(* IEC 61131-3 sources: Industry-PLC-LLM/data/PLCBEAD_repo/PLCBEAD_PLCEmbed-main/PLC-BEAD/Source/GEB/building_TIMER_2, 1 file *)

(* ---- TIMER_2.ST ---- *)
FUNCTION UDINT_TO_TIME2:TIME

	VAR_INPUT
		IN :	UDINT;
	END_VAR

	UDINT_TO_TIME2 := DINT_TO_TIME(UDINT_TO_DINT(IN));

END_FUNCTION

FUNCTION_BLOCK T_PLC_MS_block
	VAR_OUTPUT
		T_PLC_MS :	UDINT;
	END_VAR

	VAR
		PLC_TICKS_PER_SEC :	INT;
		PLC_SYS_TICK_CNT :	DINT;
	END_VAR

	VAR
		debug :	BOOL;(*Debug-Mode ON / OFF*)
		N :	INT;(*Debug-Faktor*)
		Offset :	UDINT;(*Debug-Offset*)
		temp :	DWORD := DWORD#1;(*Debug-Offset*)
		MODE :	BOOL;(*modus*)
		faktor :	UDINT;(*Systemtakt-Faktor*)
		init :	BOOL;
		v_plc_ticks_per_sec :	UDINT;
		base :	UDINT := UDINT#1000;
	END_VAR

	IF init = FALSE THEN
		v_plc_ticks_per_sec := INT_TO_UDINT(PLC_TICKS_PER_SEC);
		IF v_plc_ticks_per_sec = UDINT#1024 THEN
			faktor := UDINT#1;
			MODE := FALSE;
		ELSIF v_plc_ticks_per_sec > UDINT#0 THEN
			IF v_plc_ticks_per_sec <= base THEN
				faktor := base / v_plc_ticks_per_sec;
				MODE := FALSE;
			ELSE
				faktor := v_plc_ticks_per_sec / base;
				MODE := TRUE;
			END_IF;
		ELSE
			faktor := UDINT#1;
		END_IF;
		init := TRUE;
	END_IF;

	IF MODE THEN
		T_PLC_MS := DINT_TO_UDINT(PLC_SYS_TICK_CNT) / faktor;
	ELSE
		T_PLC_MS := DINT_TO_UDINT(PLC_SYS_TICK_CNT) * faktor;
	END_IF;

	IF debug THEN
		T_PLC_MS := (DWORD_TO_UDINT(SHL(UDINT_TO_DWORD(T_PLC_MS),N) OR SHL(temp,N)) - UDINT#1) + Offset;
	END_IF;
END_FUNCTION_BLOCK

FUNCTION DAY_OF_WEEK:INT
  VAR_INPUT
    IDATE :	UDINT;
  END_VAR

  DAY_OF_WEEK := UDINT_TO_INT((IDATE / UDINT#86400 + UDINT#3) MOD UDINT#7) + INT#01;
END_FUNCTION

FUNCTION _BYTE_TO_INT:INT
	VAR_INPUT
		IN :	BYTE;
	END_VAR

	_BYTE_TO_INT := USINT_TO_INT(BYTE_TO_USINT(IN));
END_FUNCTION

FUNCTION LEAP_OF_DATE:BOOL

	VAR_INPUT
		IDATE :	UDINT;
	END_VAR

	LEAP_OF_DATE := SHL(UDINT_TO_DWORD((IDATE + UDINT#43200) / UDINT#31557600), 30) = DWORD#16#80000000;

END_FUNCTION

FUNCTION DAY_OF_YEAR:INT
	VAR_INPUT
		IDATE :	DATE;
	END_VAR

	DAY_OF_YEAR  := UDINT_TO_INT((DATE_TO_UDINT(IDATE) / UDINT#86400) MOD UDINT#1461);
	IF DAY_OF_YEAR  > 729 THEN
		IF DAY_OF_YEAR  > 1095 THEN DAY_OF_YEAR  := DAY_OF_YEAR  - 1095; ELSE DAY_OF_YEAR  := DAY_OF_YEAR  - 729; END_IF;
	ELSIF DAY_OF_YEAR  > 364 THEN
		DAY_OF_YEAR  := DAY_OF_YEAR  - 364;
	ELSE
		DAY_OF_YEAR  := DAY_OF_YEAR  + 1;
	END_IF;
END_FUNCTION

FUNCTION DAY_OF_YEAR_UDINT:INT
	VAR_INPUT
		IDATE :	UDINT;
	END_VAR

	DAY_OF_YEAR_UDINT := UDINT_TO_INT((IDATE / UDINT#86400) MOD UDINT#1461);
	IF DAY_OF_YEAR_UDINT > 729 THEN
		IF DAY_OF_YEAR_UDINT > 1095 THEN DAY_OF_YEAR_UDINT := DAY_OF_YEAR_UDINT - 1095; ELSE DAY_OF_YEAR_UDINT := DAY_OF_YEAR_UDINT - 729; END_IF;
	ELSIF DAY_OF_YEAR_UDINT > 364 THEN
		DAY_OF_YEAR_UDINT := DAY_OF_YEAR_UDINT - 364;
	ELSE
		DAY_OF_YEAR_UDINT := DAY_OF_YEAR_UDINT + 1;
	END_IF;
END_FUNCTION

FUNCTION MONTH_OF_DATE_UDINT:INT

	VAR_INPUT
		IDATE :	UDINT;
	END_VAR

	MONTH_OF_DATE_UDINT := DAY_OF_YEAR_UDINT(IDATE);
	IF MONTH_OF_DATE_UDINT < 32 THEN
		MONTH_OF_DATE_UDINT := 1;
	ELSIF LEAP_OF_DATE(IDATE) THEN
		MONTH_OF_DATE_UDINT := (MONTH_OF_DATE_UDINT * 53 + 1668) / 1623;
	ELSE
		MONTH_OF_DATE_UDINT := (MONTH_OF_DATE_UDINT * 53 + 1700) / 1620;
	END_IF;

END_FUNCTION

FUNCTION DAY_OF_MONTH:INT
	VAR_INPUT
		IDATE :	UDINT;
	END_VAR

	DAY_OF_MONTH := DAY_OF_YEAR_UDINT(IDATE);

	IF LEAP_OF_DATE(IDATE) THEN
		CASE DAY_OF_MONTH OF
			32..60	:	DAY_OF_MONTH := DAY_OF_MONTH - 31;
			61..91	:	DAY_OF_MONTH := DAY_OF_MONTH - 60;
			92..121 :	DAY_OF_MONTH := DAY_OF_MONTH - 91;
			122..152:	DAY_OF_MONTH := DAY_OF_MONTH - 121;
			153..182:	DAY_OF_MONTH := DAY_OF_MONTH - 152;
			183..213:	DAY_OF_MONTH := DAY_OF_MONTH - 182;
			214..244:	DAY_OF_MONTH := DAY_OF_MONTH - 213;
			245..274:	DAY_OF_MONTH := DAY_OF_MONTH - 244;
			275..305:	DAY_OF_MONTH := DAY_OF_MONTH - 274;
			306..335:	DAY_OF_MONTH := DAY_OF_MONTH - 305;
			336..366:	DAY_OF_MONTH := DAY_OF_MONTH - 335;
		END_CASE;
	ELSE
		CASE DAY_OF_MONTH OF
			32..59	:	DAY_OF_MONTH := DAY_OF_MONTH - 31;
			60..90	:	DAY_OF_MONTH := DAY_OF_MONTH - 59;
			91..120 :	DAY_OF_MONTH := DAY_OF_MONTH - 90;
			121..151:	DAY_OF_MONTH := DAY_OF_MONTH - 120;
			152..181:	DAY_OF_MONTH := DAY_OF_MONTH - 151;
			182..212:	DAY_OF_MONTH := DAY_OF_MONTH - 181;
			213..243:	DAY_OF_MONTH := DAY_OF_MONTH - 212;
			244..273:	DAY_OF_MONTH := DAY_OF_MONTH - 243;
			274..304:	DAY_OF_MONTH := DAY_OF_MONTH - 273;
			305..334:	DAY_OF_MONTH := DAY_OF_MONTH - 304;
			335..365:	DAY_OF_MONTH := DAY_OF_MONTH - 334;
		END_CASE;
	END_IF;

END_FUNCTION

FUNCTION MONTH_OF_DATE:INT

	VAR_INPUT
		IDATE :	DATE;
	END_VAR

	MONTH_OF_DATE := DAY_OF_YEAR(IDATE);
	IF MONTH_OF_DATE < 32 THEN
		MONTH_OF_DATE := 1;
	ELSIF LEAP_OF_DATE(DATE_TO_UDINT(IDATE)) THEN
		MONTH_OF_DATE := (MONTH_OF_DATE * 53 + 1668) / 1623;
	ELSE
		MONTH_OF_DATE := (MONTH_OF_DATE * 53 + 1700) / 1620;
	END_IF;

END_FUNCTION

FUNCTION TIME_TO_UDINT2:UDINT
	VAR_INPUT
		X :	TIME;
	END_VAR

	TIME_TO_UDINT2 := DINT_TO_UDINT(TIME_TO_DINT(X));
END_FUNCTION

FUNCTION DT_TO_TOD2:UDINT
	VAR_INPUT
		IN :	UDINT;
	END_VAR

	DT_TO_TOD2 := (IN MOD UDINT#86400) * UDINT#1000;
END_FUNCTION

FUNCTION _DT_TO_DATE_B:UDINT

	VAR_INPUT
		_INN :	UDINT;
	END_VAR

	_DT_TO_DATE_B := (_INN / UDINT#86400) * UDINT#86400;
END_FUNCTION

FUNCTION_BLOCK TIMER_2_Block

	VAR_INPUT
		DT_IN :	UDINT;
		START :	UDINT;
		DURATION :	TIME;
		MODE :	BYTE;
		HOLIDAY  :	BOOL;
	END_VAR

	VAR_OUTPUT
		Q :	BOOL;
	END_VAR

	VAR
		last_check :	TIME := T#0s;
		dat :	UDINT;
		DAYtime :	UDINT;
		activation :	TIME;
		TX :	TIME;
		enabled :	BOOL;
		WDAY  :	INT;
		init :	BOOL;
	END_VAR

	VAR RETAIN
		run_date :	UDINT;
	END_VAR

	VAR
		T_PLC_MS :	T_PLC_MS_block;
	END_VAR

	T_PLC_MS();
	TX:= UDINT_TO_TIME(T_PLC_MS.T_PLC_MS);

	IF NOT init THEN
		init := TRUE;
		last_check := TX - t#100ms;
	END_IF;

	IF SUB_TIME(TX, last)_check < T#100ms THEN RETURN; END_IF;

	dat := _DT_TO_DATE_B(DT_IN);
	DAYtime := DT_TO_TOD2(DT_IN);
	WDAY  := DAY_OF_WEEK(dat);

	CASE _BYTE_TO_INT(MODE) OF
	1..7:
		enabled := WDAY  = _BYTE_TO_INT(MODE);
	11:
		enabled := TRUE;
	12..16:
		enabled := (dat / UDINT#86400) MOD (BYTE_TO_UDINT(MODE) - UDINT#10) = UDINT#0;
	20:
		enabled := WDAY  <= 5;
	21:
		enabled := WDAY  > 5;
	22:
		enabled := WDAY  <= 5 AND NOT holiDAY;
	23:
		enabled := WDAY  > 5 OR holiDAY;
	24:
		enabled := holiDAY;
	25:
		enabled := DAY_OF_MONTH(dat) = 1;
	26:
		enabled := DAY_OF_MONTH(dat + TIME_TO_UDINT2(t#1d)) = 1;
	27:
		enabled := DAY_OF_MONTH(dat) = 31 AND MONTH_OF_DATE_UDINT(dat) = 12;
	28:
		enabled := DAY_OF_YEAR_UDINT(dat) = 1;
	ELSE
		enabled := FALSE;
	END_CASE;

	IF enabled AND NOT Q AND DAYtime >= START AND run_date <> dat THEN
		Q := TRUE;
		activation := TX;
		run_date := dat;
	ELSIF Q AND TX - activation >= duration THEN
		Q := FALSE;
	END_IF;
	last_check := TX;

END_FUNCTION_BLOCK

PROGRAM program0
	VAR
		DT_IN :	UDINT;
		START :	UDINT;
		DURATION :	TIME;
		MODE :	BYTE;
		HOLIDAY  :	BOOL;
		Q :	BOOL;

		func_block : TIMER_2_Block;
	END_VAR
	func_block.DT_IN := DT_IN;
	func_block.START := START;
	func_block.DURATION := DURATION ;
	func_block.MODE    := MODE    ;
	func_block.HOLIDAY  := HOLIDAY;

	func_block();
	Q  := func_block.Q;
END_PROGRAM
